// TwinCAT 3 PLC project MotionPTP
// ProgramVersion: 3.1.4022.4
// libraries:
//   Tc2_MC2, * (Beckhoff Automation GmbH)
//   Tc2_Standard, * (Beckhoff Automation GmbH)
//   Tc2_System, * (Beckhoff Automation GmbH)
//   Tc2_Utilities, * (Beckhoff Automation GmbH)
//   Tc3_Module, * (Beckhoff Automation GmbH)
// project tree:
//   Function/ F_DateNow.TcPOU, F_Log.TcPOU, F_TimeNow.TcPOU
//   GVLs/ GVL_General.TcGVL
//   / PlcTask.TcTTO
//   POUs/ FB_Axis.TcPOU, MAIN.TcPOU, P_MachineLog.TcPOU
// real-time tasks:
//   TASK PlcTask: cycle T#10ms, priority 20, ADS port 350

CONFIGURATION MotionPTP
    RESOURCE PLC ON TwinCAT3
        TASK PlcTask(INTERVAL := T#10ms, PRIORITY := 20);
        PROGRAM MAIN WITH PlcTask : MAIN;
    END_RESOURCE
END_CONFIGURATION

// ---- GVLs/GVL_General.TcGVL
{attribute 'qualified_only'}
VAR_GLOBAL
	Axis1		:AXIS_REF;
	fbAxis		:FB_Axis;
	
	bPowrOn		:BOOL;
	
//----------------------HMI-----------------
	hmiPowerOn	:BOOL;
	hmiStop		:BOOL;
	hmiMoveVelo		:BOOL;
	hmiHome			:BOOL;
	hmiDummyHomeSensor		:BOOL;
	hmiSetPosition			:BOOL;
	hmiMoveRelative			:BOOL;
	hmiLActPos				:LREAL;
	hmiJogFor				:BOOL;
	hmiJogBack				:BOOL;
	hmiManualJog			:BOOL;
//-----------------------HMI-----------------

//-----------------Log---------------------
	fbLocalTime: FB_LocalSystemTime := (bEnable:= TRUE, dwCycle:= 1);
	DateTimeNow		:STRING;
	LogBufferArray: ARRAY[1..10] OF STRING := ['a','b','c','d','e','f','g','7','9','10'];
	LogBufferIndex	:INT:=1;
	sFilePath		:STRING :='C:\TempSample\';
	

//-----------------Log---------------------

	
	
END_VAR

// ---- POUs/MAIN.TcPOU
PROGRAM MAIN
VAR
	str1 : STRING;
	bTest		:BOOL;
END_VAR

//GVL_General.fbAxis();
GVL_General.fbLocalTime();

GVL_General.DateTimeNow := SYSTEMTIME_TO_STRING(GVL_General.fbLocalTime.systemTime);

str1:=   F_DateNow();



(*IF bTest THEN 
	
	F_Log('test my log function');
	bTest := FALSE;
END_IF   *)
P_MachineLog();

(*
//----------Axis---------------------
GVL_General.fbAxis.PowerOn();
GVL_General.bPowrOn :=  GVL_General.Axis1.NcToPlc.StateDWord.20;

GVL_General.fbAxis.Stop();

IF GVL_General.bPowrOn THEN 
	GVL_General.fbAxis.MoveVelocity();
	GVL_General.fbAxis.MoveRelative();	
END_IF

GVL_General.fbAxis.SetPosition();

GVL_General.hmiLActPos := GVL_General.Axis1.NcToPlc.ActPos;

GVL_General.fbAxis.SetPosition();

IF GVL_General.bPowrOn AND GVL_General.hmiManualJog THEN 
	GVL_General.fbAxis.Jog();	
END_IF
//----------Axis---------------------   *)

END_PROGRAM

// ---- Function/F_DateNow.TcPOU
FUNCTION F_DateNow : STRING
VAR_INPUT
END_VAR
VAR
END_VAR

F_DateNow := LEFT(GVL_General.DateTimeNow,10);

END_FUNCTION

// ---- POUs/P_MachineLog.TcPOU
PROGRAM P_MachineLog
VAR
	
	fbFilePuts: FB_FilePuts;
	fbFileClose: FB_FileClose;
	fbFileOpen: FB_FileOpen;
	iStep :INT;
	bFileOpened		:BOOL;
	sFileName		:STRING;
	hHandle			:UINT;	
	i				:INT; 
END_VAR

CASE iStep OF
	0:
		IF	GVL_General.LogBufferIndex >0 THEN 
			iStep := 10;
		ELSE
			iStep := 50;			
		END_IF
	10: (* check the file is open or not*)
		IF NOT bFileOpened THEN 
			iStep := 11;
		ELSE
			iStep := 20; 
		END_IF
	11:		(* try to open the file*)
		fbFileOpen(sNetId:= ,sPathName:= ,nMode:= ,ePath:= ,bExecute:= FALSE ,
					tTimeout:=T#3S ,bBusy=> ,bError=> ,nErrId=> ,hFile=> );
		IF NOT	fbFileOpen.bBusy AND NOT fbFileOpen.bError THEN 
			iStep := 12;
		END_IF
	12:	(* open the file or create the file*)
		sFileName := CONCAT(STR1:= GVL_General.sFilePath,STR2:= F_DateNow());
		sFileName := CONCAT(STR1:= sFileName,'.txt');
		fbFileOpen(sNetId:= ,sPathName:= sFileName,nMode:= FOPEN_MODEAPPEND ,ePath:= PATH_GENERIC ,bExecute:= TRUE ,
					tTimeout:=T#3S ,bBusy=> ,bError=> ,nErrId=> ,hFile=> hHandle);
		IF NOT fbFileOpen.bBusy AND NOT fbFileOpen.bError THEN 
			bFileOpened := TRUE;
			iStep := 20;
		END_IF
		
	20: (* try to write to the log file*)
		fbFilePuts(sNetId:= ,hFile:=hHandle ,sLine:=,bExecute:=FALSE,tTimeout:=T#3S,bBusy=> ,bError=> ,nErrId=> );
		IF NOT fbFilePuts.bBusy AND NOT fbFilePuts.bError THEN 
			iStep := 21;
		END_IF
	21:
		fbFilePuts(sNetId:= ,hFile:=hHandle ,sLine:=GVL_General.LogBufferArray[1],bExecute:=TRUE,tTimeout:=T#3S,bBusy=> ,bError=> ,nErrId=> );
		IF	NOT fbFilePuts.bBusy AND NOT fbFilePuts.bError THEN 
			GVL_General.LogBufferIndex := GVL_General.LogBufferIndex -1;		//???
			iStep := 22;
		END_IF
	22:
		IF	GVL_General.LogBufferIndex >1 THEN 
			FOR i := 1 TO GVL_General.LogBufferIndex - 1 DO
				GVL_General.LogBufferArray[i] := GVL_General.LogBufferArray[i + 1];
			END_FOR
			iStep := 0;
		ELSE 
			iStep := 50;
		END_IF
	
	50:
		fbFileClose(sNetId:= ,hFile:= fbFileOpen.hFile,bExecute:=FALSE,tTimeout:=T#3S ,	bBusy=> ,bError=> ,nErrId=> );
		IF NOT fbFileClose.bBusy THEN 
			IF NOT fbFileClose.bError THEN 
				iStep:= 51;
			END_IF
		END_IF
		
	51:
		fbFileClose(sNetId:= ,hFile:=fbFileOpen.hFile,bExecute:=TRUE,tTimeout:=T#3S,bBusy=> ,bError=> ,nErrId=> );
		
		IF NOT fbFileClose.bBusy AND NOT fbFileClose.bError THEN 
			bFileOpened := FALSE;
			iStep := 0;
		ELSE 
			iStep := 999;
		END_IF
	999:
		;
END_CASE

END_PROGRAM

// ---- POUs/FB_Axis.TcPOU
FUNCTION_BLOCK FB_Axis
VAR_INPUT
	//axis		:AXIS_REF;
	
END_VAR
VAR_OUTPUT
END_VAR
VAR	
	fbPower: MC_Power;
	
	fbMoveVelocity: MC_MoveVelocity;
	fbStop: MC_Stop;
	fbMoveRelative: MC_MoveRelative;
	fbHome: MC_Home;
	fbJog: MC_Jog;
	fbSetPosition: MC_SetPosition;
	fbReset: MC_Reset;
	rTrig: R_TRIG;
END_VAR

METHOD Homing : BOOL
VAR_INPUT
END_VAR


fbHome(Axis:=GVL_General.Axis1,Execute:=GVL_General.hmiHome,Position:=0,HomingMode:= ,BufferMode:= ,Options:= , 
	bCalibrationCam:= GVL_General.hmiDummyHomeSensor,Done=> ,Busy=> ,Active=> ,CommandAborted=> ,Error=> ,ErrorID=> );
END_METHOD

METHOD Jog : BOOL
VAR_INPUT
END_VAR
fbJog(
	Axis:=GVL_General.Axis1 , 
	JogForward:=GVL_General.hmiJogFor , 
	JogBackwards:= GVL_General.hmiJogBack, 
	Mode:= MC_JOGMODE_CONTINOUS, 
	Position:= , 
	Velocity:= 10, 
	Acceleration:= , 
	Deceleration:= , 
	Jerk:= , 
	Done=> , 
	Busy=> , 
	Active=> , 
	CommandAborted=> , 
	Error=> , 
	ErrorID=> );
END_METHOD

METHOD MoveRelative : BOOL
VAR_INPUT
END_VAR
fbMoveRelative(
	Axis:= GVL_General.Axis1, 
	Execute:=GVL_General.hmiMoveRelative, 
	Distance:= 30, 
	Velocity:= 1, 
	Acceleration:= , 
	Deceleration:= , 
	Jerk:= , 
	BufferMode:= , 
	Options:= , 
	Done=> , 
	Busy=> , 
	Active=> , 
	CommandAborted=> , 
	Error=> , 
	ErrorID=> );
	
IF GVL_General.hmiMoveRelative THEN 
	GVL_General.hmiMoveRelative	:= FALSE;
END_IF
END_METHOD

METHOD MoveVelocity : BOOL
VAR_INPUT
END_VAR
fbMoveVelocity(Axis:=GVL_General.Axis1, 
	Execute:=GVL_General.hmiMoveVelo, 
	Velocity:=500, 
	Acceleration:=, 
	Deceleration:= , 
	Jerk:= , 
	Direction:=MC_Direction.MC_Positive_Direction, 
	BufferMode:= , 
	Options:= , 
	InVelocity=> , 
	Busy=> , 
	Active=> , 
	CommandAborted=> , 
	Error=> , 
	ErrorID=> );
	
IF	GVL_General.hmiMoveVelo THEN 
	GVL_General.hmiMoveVelo := FALSE;
END_IF
END_METHOD

METHOD PowerOn : BOOL
VAR_INPUT
END_VAR

//F_Log('Axis Power On');

fbPower(
	Axis:=GVL_General.Axis1 , 
	Enable:= GVL_General.hmiPowerOn,
	Enable_Positive:=TRUE , 
	Enable_Negative:= TRUE, 
	Override:= , 
	BufferMode:= , 
	Options:= ,
	Status=> , 
	Busy=> , 
	Active=> , 
	Error=> , 
	ErrorID=> );
END_METHOD

METHOD SetPosition : BOOL
VAR_INPUT
END_VAR
fbSetPosition(
	Axis:=GVL_General.Axis1, 
	Execute:=GVL_General.hmiSetPosition, 
	Position:=0, 
	Mode:= , 
	Options:= , 
	Done=> , 
	Busy=> , 
	Error=> , 
	ErrorID=> );
	
IF	GVL_General.hmiSetposition THEN 
	GVL_General.hmiSetposition := FALSE;
END_IF
END_METHOD

METHOD Stop : BOOL
VAR_INPUT
END_VAR
rTrig(CLK:=GVL_General.hmiStop , Q=> );

fbStop(Axis:= GVL_General.Axis1,Execute:=rTrig.Q, Deceleration:= , 
	Jerk:= ,Options:= ,Done=> ,Busy=> ,Active=> ,CommandAborted=> ,	Error=> , 
	ErrorID=> );
	
IF GVL_General.hmiStop  THEN 
	GVL_General.hmiStop	:= FALSE;
END_IF
END_METHOD

END_FUNCTION_BLOCK

// ---- Function/F_Log.TcPOU
FUNCTION F_Log : bool
VAR_INPUT
	str1		:STRING;
END_VAR
VAR
END_VAR

GVL_General.LogBufferIndex := GVL_General.LogBufferIndex + 1;

GVL_General.LogBufferArray[GVL_General.LogBufferIndex] := str1;

END_FUNCTION

// ---- Function/F_TimeNow.TcPOU
FUNCTION F_TimeNow : STRING
VAR
	
END_VAR



F_TimeNow := RIGHT(GVL_General.DateTimeNow,12);

END_FUNCTION
